Staubli VAL3: PulesAdd.pgx

public program PulesAdd()
  local num l_nPulse
begin
  for l_nPulse=0 to 99 step 1
    delay(0.02)
    fOut0=true
    fOut0=false

  endFor

end
